FUNCTION NetEv2NetEv (* Manipulate NetEv *)
  (* Standard: 61499-1 *)
  (* Version 1.0, 2025-10-24, Franz Höpfinger *)
  PACKAGE isobus::PGN;
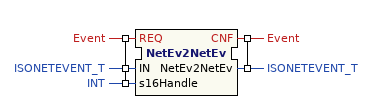
  EVENT_INPUT
    REQ WITH IN, s16Handle;
  END_EVENT
  EVENT_OUTPUT
    CNF WITH NetEv2NetEv;
  END_EVENT
  VAR_INPUT
    IN : isobus::pgn::ISONETEVENT_T; (* ISONETEVENT_T Input *)
    s16Handle : INT; (* Network member handle of the CF / user (event source CF handle) *)
  END_VAR
  VAR_OUTPUT
    NetEv2NetEv : isobus::pgn::ISONETEVENT_T;
  END_VAR
  BODY IN ST:
PACKAGE isobus::PGN;

(* Manipulate NetEv *)
FUNCTION NetEv2NetEv : ISONETEVENT_T

VAR_INPUT
	IN : ISONETEVENT_T; // ISONETEVENT_T Input
	s16Handle : INT; // Network member handle of the CF / user (event source CF handle)
END_VAR

NetEv2NetEv := IN;
NetEv2NetEv.s16Handle := s16Handle;

END_FUNCTION
  END_BODY
END_FUNCTION
